PROGRAM P_CraneSim
VAR
	fbCraneSim		: FB_CraneSimulator;
	bSimulatorOn			: BOOL;
	fValeInput				: LREAL;
	fCylinderPosition		: LREAL;
	fPistonSidePressure			: LREAL;
	fRodSidePressure		: LREAL;
END_VAR

fbCraneSim(
	ssMethodType := BOOL_TO_SINT(bSimulatorOn),
	uDCV := fValeInput,
	xm => fCylinderPosition,
	ppbar => fPistonSidePressure,
	prbar => fRodSidePressure
);

END_PROGRAM

(* stored: Version 1.1.0.1, ProductVersion 3.1.4024.12
   POU P_CraneSim: Id {abd16a88-c182-46f2-9f6f-a5822b2fe25a}, SpecialFunc None *)
